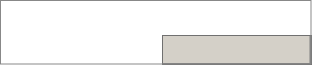
VISUALIZATION Visualization  // 312x65
    Button (162,35 150x30)
END_VISUALIZATION

(* stored: Version 1.1.0.1, ProductVersion 3.1.4024.4
   Visu Visualization: Id {67935ccf-fd1e-4967-bafd-27e006ff6adc} *)
